TYPE T_ASTRO_POLAR_MOTION :
STRUCT
	x : LREAL := 0.0;
	y : LREAL := 0.0;
END_STRUCT
END_TYPE

(* stored: Version 1.1.0.1, ProductVersion 3.1.4024.11
   DUT T_ASTRO_POLAR_MOTION: Id {f8dec1da-498d-4142-8fcd-3a200b59e940} *)
